// TIA Portal V20 export
TYPE "LWONIK_typePhmiMode"
// stored: Access Published
   STRUCT
      estop : Bool;
      enable : Bool;
      reset : Bool;
      PhmiForcedDisconnection : Bool;
   END_STRUCT;
END_TYPE
